KUKA KRL program: chk_w3_wechs_ok.src

&ACCESS RV1
&REL 5
&COMMENT GUN C2
DEF chk_w3_wechs_ok( )

; VERIFICAÇÃO DE FERRAMENTA: C2

$TIMER[10] = 0
$TIMER_STOP[10] = FALSE

wait for (($IN[585]) and ($IN[577]) and ($in[161]) and (($in[177]) or (NOT ($in[177]) and $in[3320])) and ($in[193]) and ($in[201]) and ($in[209]) and (not $IN[169]) and ($in[185]) AND ($in[219]))

$TIMER_STOP[10] = TRUE
$TIMER[10] = 0

;//---- End -------
;Diag_Appl(#Off,5)

END
